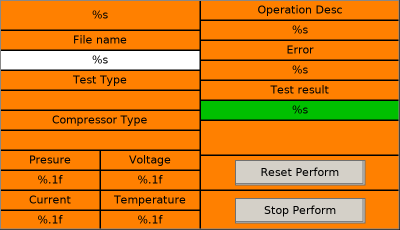
VISUALIZATION vSmallChamber_v2_WEB  // 400x230
VAR_IN_OUT
	stParams : stParamsChamber;
	fbChamber : fbChamber;
	stControl : stControl;
END_VAR
    Rectangle (200,155 200x35)
    Rectangle (200,120 200x35)
    Rectangle (0,50 200x20), "%s", text variable: fbChamber.sTestName
        OnMouseClick: write the text variable via VisuDialogs.Keypad
    Rectangle (0,30 200x20), "File name"
    Rectangle (0,90 200x20), text list: 'txlTestTypes', text index: fbChamber.stControl.iSetTest
    Rectangle (0,70 200x20), "Test Type"
    Rectangle (0,110 200x20), "Compressor Type"
    Rectangle (0,130 200x20), text list: 'txlCompresorTypes', text index: fbChamber.stParams.iCompresorType
    Rectangle (0,150 100x20), "Presure"
    Rectangle (100,150 100x20), "Voltage"
    Rectangle (0,170 100x20), "%.1f", text variable: fbChamber.stInOuts.rPressure
    Rectangle (100,170 100x20), "%.1f", text variable: fbChamber.stInOuts.rVoltage
    Rectangle (0,190 100x20), "Current"
    Rectangle (0,210 100x20), "%.1f", text variable: fbChamber.stInOuts.rVoltage
    Rectangle (200,0 200x20), "Operation Desc"
    Rectangle (200,20 200x20), "%s", text variable: fbChamber.sStepDescription
    Rectangle (200,80 200x20), "Test result"
    Rectangle (200,100 200x20), "%s", text variable: stControl.sTestResult, colour toggle: stControl.sTestResult <> 'DONE'
    Rectangle (200,40 200x20), "Error"
    Rectangle (200,60 200x20), "%s", text variable: stParams.sErrorDescription
    Rectangle (0,0 200x30), "%s", text variable: stParams.sChamberName
    Button (235,160 130x25), "Reset Perform"
        OnMouseClick: toggle stControl.bResetChamber
    Rectangle (100,210 100x20), "%.1f", text variable: fbChamber.stInOuts.rTemperature
    Rectangle (100,190 100x20), "Temperature"
    Rectangle (200,190 200x40)
    Button (235,198 130x25), "Stop Perform"
        OnMouseClick: toggle stControl.bStopPerform
END_VISUALIZATION

(* stored: Version 1.1.0.1, ProductVersion 3.1.4024.12
   Visu vSmallChamber_v2_WEB: Id {410ae35c-6aad-45ee-b616-bad81ca0afd8} *)
